# B&R Automation Studio project Zbiorniki_user
Automation Studio 4.9

## Configuration X20CP1584

CPU X20CP1584, AutomationRuntime J4.93, Build 4.1.2, Safety 0.0, Vc V4.34.3

### Task classes (Cpu.sw)
```
Cyclic#1:
  ClockSigna <- Wizualizacja.ClockSignal.prg
Cyclic#4:
  Tanks <- Sterowanie.Tanks.prg
  Recipies <- Sterowanie.Recipies.prg
  Visibility <- HelpingFunctions.Visibility.prg
Cyclic#8:
  Alarms <- Alarms.Alarms.prg
Binaries: arsvcreg, TCData, TCLang, OpcUaSrv, udbdef, mvLoader, iomap, Role, arconfig, asfw, ashwac, sysconf, User, TankAlarm, ashwd
Libraries: standard, MpAlarmX, MpBase, astime, runtime, MpServer, MpWebXs, AsArSdm, dataobj, fileio, sys_lib, asieccon, arssl, aruser
```

### Hardware
```
X20CP1584 : X20CP1584 v1.10.0.0
  Connector IF2:
    ActivateDevice = 1
  Connector IF3:
    DNAConfiguration = manual
  ConfigurationID = CaseWeek_user_X20CP1584
  UserPartitionSize = 0
  Simulation = 1
  FileDevice1
  FileDeviceName1 = USER
  FileDevicePath1 = USER_PATH
  ActivateOpcUa = 1
  OpcUaInformationModels_PV_Version = 1
```

### TankAlarm.mpalarmxcore - X20CP1584/mappServices/Tank/TankAlarm.mpalarmxcore
```
Element MpLinkTankAlarmXCore (Type=mpalarmxcore)
  mapp.AlarmX.Core.Configuration:
    [0]:
      Name = TankLevelHigh
      Message = Tank level is high!
      Behavior = PersistentAlarm
    [1]:
      Name = PressureLevelHigh
      Message = Pressure level is high!
      Behavior = PersistentAlarm
    [2]:
      Name = PresureLevelCritical
      Message = The pressure level is critical! Turning on the vales!
      Severity = 5
      Behavior = PersistentAlarm
```

## Logical view

Binary libraries used (declarations not repeated): operator, runtime, astime, AsIecCon, standard, MpAlarmX, MpBase, MpServer, MpWebXs 5.24.5, AsArSdm

### Package Logical/Libraries - Global libraries

- Visualisation Logical/mappView (not shown)

### mappingVariables.var
```iecst
(*Zmienne które sa uzywane przez symulacje. Nalezy je przypisac do zmiennych w programie sterujacym*)
VAR
	gZb1_poziom : INT; (*Poziom cieczy w zbiorniku 1*)
	gZb2_poziom : INT; (*Poziom cieczy w zbiorniku 2*)
	gZb3_poziom : INT; (*Poziom cieczy w zbiorniku 3*)
	gZb1_zawor : BOOL; (*0 - zawor zamkniety, 1 - zawor otwarty*)
	gZb2_zawor : BOOL; (*0 - zawor zamkniety, 1 - zawor otwarty*)
	gZb3_zawor_lewy : INT; (*% otwarcia zaworu lewego (0-100)*)
	gZb3_zawor_prawy : INT; (*% otwarcia zaworu prawego (0-100)*)
	gZb3_zawor_glowny : BOOL; (*0 - zawor zamkniety, 1 - zawor otwarty*)
	gMieszadlo : BOOL; (*0 - mieszadlo wylaczone, 1- mieszadlo wlaczone*)
	START : BOOL;
	STOP : BOOL;
	PAUSE : BOOL;
	MIESZANIE : BOOL;
	NOT_STOP : BOOL;
	MANUAL : BOOL;
END_VAR
```

### Program Logical/Sterowanie/Tanks (IEC)

#### Main.st
```iecst
PROGRAM _INIT

END_PROGRAM
PROGRAM _CYCLIC

END_PROGRAM

PROGRAM _EXIT

END_PROGRAM
```

### Program Logical/Sterowanie/ControlTanks (IEC)

#### Main.st - Init, cyclic, exit code
```iecst
PROGRAM _INIT
	gZb1_poziom := 0;
	gZb1_zawor := 0;
	gZb2_poziom := 0;
	gZb2_zawor := 0;
	gZb3_poziom := 0;
	gZb3_zawor_glowny := 0;
	gZb3_zawor_lewy := 0;
	gZb3_zawor_prawy := 0;
	gMieszadlo := 0;
	Mieszanie := 0;
	krok := 0;
	timer_mieszania.IN := FALSE;
	timer_uruchomiony := FALSE;
	before_MANUAL := FALSE;

	UstawieniaDomyslne;
END_PROGRAM

PROGRAM _CYCLIC
	IF MANUAL THEN
		ObslugaManual;
	ELSE
		ObslugaAuto;
	END_IF;

	before_MANUAL := MANUAL;
	ObslugaStop;
END_PROGRAM

PROGRAM _EXIT
	ResetWyjsc;
END_PROGRAM
```

#### Variables.var - Local variables
```iecst
VAR
	before_MANUAL : BOOL;
	krok : USINT;
	Mieszanie : BOOL;
	timer_mieszania : TON;
	czas_mieszania : TIME := T#5s;
	aktywny : BOOL;

	zawor1_otwarcie : BOOL := TRUE;
	zawor2_otwarcie : BOOL := TRUE;
	zawor3_glowny_otwarcie : BOOL := TRUE;

	zawor3_lewy_aktywny : BOOL := TRUE;
	zawor3_prawy_aktywny : BOOL := TRUE;
	zawor3_lewy_otwarcie : INT := 50;
	zawor3_prawy_otwarcie : INT := 50;

	default_lewy_procent : INT := 50;
	default_prawy_procent : INT := 50;

	tolerancja_poziom : INT := 100;
	timer_uruchomiony : BOOL := FALSE;
	max_poziom : INT := 10000;
	poziom_95_procent : INT := 9500;
	poziom_80_procent : INT := 8000;
END_VAR
```

#### UstawieniaDomyslne.st
```iecst
ACTION UstawieniaDomyslne:
	zawor1_otwarcie := TRUE;
	zawor2_otwarcie := TRUE;
	zawor3_glowny_otwarcie := TRUE;
	zawor3_lewy_aktywny := TRUE;
	zawor3_prawy_aktywny := TRUE;
	zawor3_lewy_otwarcie := default_lewy_procent;
	zawor3_prawy_otwarcie := default_prawy_procent;
END_ACTION
```

#### ResetWyjsc.st
```iecst
ACTION ResetWyjsc:
	gZb1_zawor := 0;
	gZb2_zawor := 0;
	gZb3_zawor_glowny := 0;
	gZb3_zawor_lewy := 0;
	gZb3_zawor_prawy := 0;
	gMieszadlo := 0;
END_ACTION
```

#### ZabezpieczeniaPoziomow.st
```iecst
ACTION ZabezpieczeniaPoziomow:
	IF gZb1_poziom >= poziom_95_procent THEN
		gZb1_zawor := 0;
	END_IF;

	IF gZb2_poziom >= poziom_95_procent THEN
		gZb2_zawor := 0;
	END_IF;

	IF gZb3_poziom >= max_poziom THEN
		gZb3_zawor_prawy := 0;
		gZb3_zawor_lewy := 0;
	END_IF;
END_ACTION
```

#### ObslugaManual.st
```iecst
ACTION ObslugaManual:
	timer_mieszania.IN := FALSE;
	timer_uruchomiony := FALSE;
	ZabezpieczeniaPoziomow;
END_ACTION
```

#### ObslugaAuto.st
```iecst
ACTION ObslugaAuto:
	IF before_MANUAL AND NOT MANUAL THEN
		krok := 0;
		timer_mieszania.IN := FALSE;
		timer_uruchomiony := FALSE;
		UstawieniaDomyslne;
	END_IF;

	aktywny := NOT PAUSE;
	Mieszanie := MIESZANIE;
	timer_mieszania();

	ResetWyjsc;

	CASE krok OF
		0: KrokStop;
		1: KrokNapelnianie12;
		2: KrokNapelnianie3;
		3: KrokMieszanie;
		4: KrokOprozniane;
		5: KrokWyrownywanie;
	END_CASE;

	IF PAUSE THEN
		ResetWyjsc;
	END_IF;
END_ACTION
```

#### KrokStop.st
```iecst
ACTION KrokStop:
	timer_mieszania.IN := FALSE;
	timer_uruchomiony := FALSE;

	IF aktywny AND START AND NOT STOP THEN
		IF ABS(gZb1_poziom - gZb2_poziom) > tolerancja_poziom THEN
			krok := 5;
		ELSE
			IF gZb1_poziom >= poziom_80_procent AND gZb2_poziom >= poziom_80_procent THEN
				krok := 2;
			ELSE
				krok := 1;
			END_IF;
		END_IF;
	END_IF;
END_ACTION
```

#### KrokNapelnianie12.st
```iecst
ACTION KrokNapelnianie12:
	IF aktywny THEN
		IF gZb1_poziom >= poziom_80_procent AND gZb2_poziom >= poziom_80_procent THEN
			krok := 2;
		ELSE
			IF zawor1_otwarcie AND gZb1_poziom < poziom_80_procent AND gZb1_poziom < poziom_95_procent THEN
				gZb1_zawor := 1;
			END_IF;
			IF zawor2_otwarcie AND gZb2_poziom < poziom_80_procent AND gZb2_poziom < poziom_95_procent THEN
				gZb2_zawor := 1;
			END_IF;
		END_IF;

		gZb3_zawor_lewy := 0;
		gZb3_zawor_prawy := 0;
	END_IF;
END_ACTION
```

#### KrokNapelnianie3.st
```iecst
ACTION KrokNapelnianie3:
	IF aktywny THEN
		UstawZaworyZbiornika3;

		IF gZb3_poziom >= poziom_80_procent AND NOT Mieszanie THEN
			krok := 4;
		END_IF;

		IF gZb3_poziom >= max_poziom AND Mieszanie THEN
			krok := 3;
			timer_uruchomiony := FALSE;
		END_IF;
	END_IF;
END_ACTION
```

#### UstawZaworyZbiornika3.st
```iecst
ACTION UstawZaworyZbiornika3:
	IF zawor3_prawy_aktywny AND zawor3_prawy_otwarcie > 0 THEN
		gZb3_zawor_prawy := zawor3_prawy_otwarcie;
	ELSE
		gZb3_zawor_prawy := 0;
	END_IF;

	IF zawor3_lewy_aktywny AND zawor3_lewy_otwarcie > 0 THEN
		gZb3_zawor_lewy := zawor3_lewy_otwarcie;
	ELSE
		gZb3_zawor_lewy := 0;
	END_IF;
END_ACTION
```

#### KrokMieszanie.st
```iecst
ACTION KrokMieszanie:
	IF aktywny THEN
		gMieszadlo := 1;

		IF NOT timer_uruchomiony THEN
			timer_mieszania.IN := TRUE;
			timer_mieszania.PT := czas_mieszania;
			timer_uruchomiony := TRUE;
		END_IF;

		IF timer_mieszania.Q THEN
			timer_mieszania.IN := FALSE;
			timer_uruchomiony := FALSE;
			krok := 4;
		END_IF;
	ELSE
		timer_mieszania.IN := FALSE;
	END_IF;
END_ACTION
```

#### KrokOprozniane.st
```iecst
ACTION KrokOprozniane:
	IF aktywny THEN
		IF zawor3_glowny_otwarcie THEN
			gZb3_zawor_glowny := 1;
		END_IF;

		IF gZb3_poziom = 0 THEN
			krok := 0;
		END_IF;
	END_IF;
END_ACTION
```

#### KrokWyrownywanie.st
```iecst
ACTION KrokWyrownywanie:
	IF aktywny THEN
		IF gZb1_poziom > gZb2_poziom + tolerancja_poziom THEN
			gZb1_zawor := 0;
			IF zawor2_otwarcie AND gZb2_poziom < poziom_95_procent THEN
				gZb2_zawor := 1;
			END_IF;
		ELSIF gZb2_poziom > gZb1_poziom + tolerancja_poziom THEN
			gZb2_zawor := 0;
			IF zawor1_otwarcie AND gZb1_poziom < poziom_95_procent THEN
				gZb1_zawor := 1;
			END_IF;
		ELSE
			gZb1_zawor := 0;
			gZb2_zawor := 0;

			IF gZb1_poziom >= poziom_80_procent AND gZb2_poziom >= poziom_80_procent THEN
				krok := 2;
			ELSE
				krok := 1;
			END_IF;
		END_IF;
	END_IF;
END_ACTION
```

#### ObslugaStop.st
```iecst
ACTION ObslugaStop:
	IF STOP THEN
		krok := 0;
		timer_mieszania.IN := FALSE;
		timer_uruchomiony := FALSE;

		IF MANUAL THEN
			ResetWyjsc;
		END_IF;
	END_IF;
END_ACTION
```

### Program Logical/Sterowanie/Recipies

#### Variables.var
```iecst
VAR
	before_MANUAL : BOOL;
	krok : USINT;
	Mieszanie : BOOL;
	timer_mieszania : TON;
	czas_mieszania : TIME := T#5s;
	aktywny : BOOL;

	zawor1_otwarcie : BOOL;
	zawor2_otwarcie : BOOL;
	zawor3_glowny_otwarcie : BOOL;
	zawor3_lewy_otwarcie : INT := 100;
	zawor3_prawy_otwarcie : INT := 100;

	tolerancja_poziom : INT := 100;
   	timer_uruchomiony : BOOL := FALSE;
	max_poziom : INT := 10000;
	poziom_95_procent : INT := 9500;
END_VAR
```

#### Main.st
```iecst
PROGRAM _INIT
    // Inicjalizacja poziomów zbiorników
	gZb1_poziom := 0;
	gZb1_zawor := 0;
	gZb2_poziom := 0;
	gZb2_zawor := 0;

	gZb3_poziom := 0;
	gZb3_zawor_glowny := 0;
	gZb3_zawor_lewy := 0;
	gZb3_zawor_prawy := 0;

	gMieszadlo := 0;

	Mieszanie:= 0;

	// Inicjalizacja stanu
	krok := 0;
	timer_mieszania.IN := FALSE;
END_PROGRAM

PROGRAM _CYCLIC
    // Sprawdzenie trybu manualnego
	IF MANUAL THEN
		// W trybie manualnym nie nadpisujemy wyjść automatyką
		// Wyłączenie timera w trybie manualnym
		timer_mieszania.IN := FALSE;
		timer_uruchomiony := FALSE;

		// ZABEZPIECZENIE: Automatyczne wyłączenie zaworów przy 95% poziomu
		IF gZb1_poziom >= poziom_95_procent THEN
			gZb1_zawor := 0;
		END_IF;

		IF gZb2_poziom >= poziom_95_procent THEN
			gZb2_zawor := 0;
		END_IF;

	ELSE
		// Tryb automatyczny - sprawdzenie czy wyszliśmy z trybu manualnego
		IF before_MANUAL AND NOT MANUAL THEN
			krok := 0;
			timer_mieszania.IN := FALSE;
			timer_uruchomiony := FALSE;
		END_IF;

		aktywny := NOT PAUSE;
		Mieszanie := MIESZANIE;

		// Wywołanie timera zawsze (poza trybem manualnym)
		timer_mieszania();

		// Domyślne ustawienie wyjść na 0 (bezpieczne)
		gZb1_zawor := 0;
		gZb2_zawor := 0;
		gZb3_zawor_glowny := 0;
		gZb3_zawor_lewy := 0;
		gZb3_zawor_prawy := 0;
		gMieszadlo := 0;

		// Maszyna stanów - zawsze wykonywana, ale akcje warunkowane przez 'aktywny'
		CASE krok OF
			0: // STOP
				// Reset timera przy wejściu do STOP
				timer_mieszania.IN := FALSE;
				timer_uruchomiony := FALSE;

				// Przejście do wyrównywania poziomów po START (jeśli potrzebne)
				IF aktywny AND START AND NOT STOP THEN
					IF ABS(gZb1_poziom - gZb2_poziom) > tolerancja_poziom THEN
						krok := 5;
					ELSE
						IF gZb1_poziom >= 8000 AND gZb2_poziom >= 8000 THEN
							krok := 2;
						ELSE
							krok := 1;
						END_IF;
					END_IF;
				END_IF;

			1: // NAPEŁNIANIE ZBIORNIKÓW 1 i 2
				IF aktywny THEN
					IF gZb1_poziom >= 8000 AND gZb2_poziom >= 8000 THEN
						krok := 2;
					ELSE
						IF zawor1_otwarcie > 0 AND gZb1_poziom < 8000 AND gZb1_poziom < poziom_95_procent THEN
							gZb1_zawor := 1;
						END_IF;
						IF zawor2_otwarcie > 0 AND gZb2_poziom < 8000 AND gZb2_poziom < poziom_95_procent THEN
							gZb2_zawor := 1;
						END_IF;
					END_IF;

					gZb3_zawor_lewy := 0;
					gZb3_zawor_prawy := 0;
				END_IF;

			2: // NAPEŁNIANIE ZBIORNIKA 3
				IF aktywny THEN
					gZb3_zawor_prawy := zawor3_prawy_otwarcie;
					gZb3_zawor_lewy := zawor3_lewy_otwarcie;

					IF gZb3_poziom >= 8000 AND NOT Mieszanie THEN
						krok := 4;
					END_IF;

					IF gZb3_poziom >= 10000 AND Mieszanie THEN
						krok := 3;
						// Reset flagi timera przy wejściu do kroku mieszania
						timer_uruchomiony := FALSE;
					END_IF;
				END_IF;

			3: // MIESZANIE ZBIORNIKA 3
				IF aktywny THEN
					// Włączenie mieszadła
					gMieszadlo := 1;

					// Uruchomienie timera tylko raz przy wejściu do kroku
					IF NOT timer_uruchomiony THEN
						timer_mieszania.IN := TRUE;
						timer_mieszania.PT := czas_mieszania;
						timer_uruchomiony := TRUE;
					END_IF;

					// Sprawdzenie końca mieszania
					IF timer_mieszania.Q THEN
						timer_mieszania.IN := FALSE;
						timer_uruchomiony := FALSE;
						krok := 4;
					END_IF;

				ELSE
					// Podczas pauzy: Wyłącz timer ale zachowaj jego stan
					timer_mieszania.IN := FALSE;
				END_IF;

			4: // OPRÓŻNIANIE ZBIORNIKA 3
				IF aktywny THEN
					IF zawor3_glowny_otwarcie > 0 THEN
						gZb3_zawor_glowny := 1;
					END_IF;

					IF gZb3_poziom = 0 THEN
						krok := 0;
					END_IF;
				END_IF;

			5: // WYRÓWNYWANIE POZIOMÓW ZBIORNIKÓW 1 i 2
				IF aktywny THEN
					IF gZb1_poziom > gZb2_poziom + tolerancja_poziom THEN
						gZb1_zawor := 0;
						IF zawor2_otwarcie > 0 AND gZb2_poziom < poziom_95_procent THEN
							gZb2_zawor := 1;
						END_IF;
					ELSIF gZb2_poziom > gZb1_poziom + tolerancja_poziom THEN
						gZb2_zawor := 0;
						IF zawor1_otwarcie > 0 AND gZb1_poziom < poziom_95_procent THEN
							gZb1_zawor := 1;
						END_IF;
					ELSE
						gZb1_zawor := 0;
						gZb2_zawor := 0;

						IF gZb1_poziom >= 8000 AND gZb2_poziom >= 8000 THEN
							krok := 2;
						ELSE
							krok := 1;
						END_IF;
					END_IF;
				END_IF;

		END_CASE;

		// Jeśli pauza, nadpisz wszystkie wyjścia na 0 (dla bezpieczeństwa)
		IF PAUSE THEN
			gZb1_zawor := 0;
			gZb2_zawor := 0;
			gZb3_zawor_glowny := 0;
			gZb3_zawor_lewy := 0;
			gZb3_zawor_prawy := 0;
			gMieszadlo := 0;
			// Timer pozostaje w stanie pauzy (nie resetujemy go)
		END_IF;

	END_IF;

	// Zapamiętanie stanu MANUAL dla wykrycia przejścia
	before_MANUAL := MANUAL;

	// Globalne sprawdzenie STOP - działa zawsze, nawet w trybie manualnym
	IF STOP THEN
		krok := 0;
		timer_mieszania.IN := FALSE;
		timer_uruchomiony := FALSE;

		IF MANUAL THEN
			gZb_zawor := 0;
			gZb2_zawor := 0;
			gZb3_zawor_glowny := 0;
			gZb3_zawor_lewy := 0;
			gZb3_zawor_prawy := 0;
			gMieszadlo := 0;
		END_IF;
	END_IF;

END_PROGRAM

PROGRAM _EXIT
    // Bezpieczne wyłączenie wszystkich urządzeń
	gZb1_zawor := 0;
	gZb2_zawor := 0;
	gZb3_zawor_glowny := 0;
	gZb3_zawor_lewy := 0;
	gZb3_zawor_prawy := 0;
	gMieszadlo := 0;
END_PROGRAM
```

### Program Logical/Alarms/Alarms

#### Variables.var
```iecst
VAR
	MpAlarmXCore_0 : MpAlarmXCore;
	ALARM_TANK_HIGH : INT := 9000;
END_VAR
```

#### Main.st
```iecst
PROGRAM _INIT
	(* Insert code here *)
	 MpAlarmXCore_0(MpLink := ADR(MpLinkTankAlarmXCore) , Enable := TRUE);
END_PROGRAM

PROGRAM _CYCLIC
	MpAlarmXCore_0(MpLink := ADR(MpLinkTankAlarmXCore) , Enable := TRUE);
	IF gZb1_poziom > ALARM_TANK_HIGH OR gZb2_poziom > ALARM_TANK_HIGH THEN
		MpAlarmXSet(MpLinkTankAlarmXCore, 'TankLevelHigh');
	ELSE
		MpAlarmXReset(MpLinkTankAlarmXCore, 'TankLevelHigh');
	END_IF

END_PROGRAM

PROGRAM _EXIT
	(* Insert code here *)
	MpAlarmXCore_0(Enable := FALSE);
END_PROGRAM
```

### Program Logical/HelpingFunctions/Visibility (IEC)

#### Main.st
```iecst
PROGRAM _INIT
	(* Insert code here *)
	MANUAL := FALSE;
END_PROGRAM

PROGRAM _CYCLIC
	// The variables used here are only for helping purposes, they are here so we avoid being lost in the expressions.
	NOT_STOP := NOT STOP;
	IF STOP THEN
		START := FALSE;
	END_IF

END_PROGRAM

PROGRAM _EXIT
	(* Insert code here *)

END_PROGRAM
```

Listed in the project but not available here: Logical/Global.typ, Logical/Global.var, Logical/Wizualizacja, Logical/Sterowanie/ControlTanks/Types.typ
